{attribute 'strict'}
TYPE E_FixtureStateMeasurementDataExchange :
(
	FIXTURE_MEASURE_DATA_EXCHANGING_WAIT_FOR_BUSY 		:= 0,
	FIXTURE_MEASURE_DATA_EXCHANGING_WAIT_FOR_FISNISH 	:= 10,
	FIXTURE_MEASURE_DATA_EXCHANGING_PROCCESS_RESULTS 	:= 20,
	FIXTURE_MEASURE_DATA_EXCHANGING_DONE				:= 30
);
END_TYPE

(* stored: Version 1.1.0.1, ProductVersion 3.1.4024.9
   DUT E_FixtureStateMeasurementDataExchange: Id {81decc9f-867d-4363-b28d-f0b680c02d8d} *)
